// TIA Portal V16 export
// export: Created 2024-12-03T15:41:45.8171192Z, ExportSetting WithReadOnly, DisplayName Totally Integrated Automation Portal, DisplayVersion V16 Update 6, DisplayName TIA Portal Version Control Interface, DisplayVersion V16 Update 2, DisplayName TIA Portal Openness, DisplayVersion V16 Update 6, DisplayName TIA Portal Teamcenter Gateway, DisplayVersion V16, DisplayName SINAMICS Startdrive Advanced, DisplayVersion V16 Update 5, DisplayName SINAMICS Startdrive G130, G150, S120, S150, SINAMICS MV, S210, DisplayVersion V16 Update 5, DisplayName SINAMICS Startdrive G110M, G120, G120C, G120D, G120P, G115D, DisplayVersion V16 Update 5, DisplayName STEP 7 Professional, DisplayVersion V16 Update 6, DisplayName STEP 7 Safety, DisplayVersion V16, DisplayName WinCC Advanced / Unified PC, DisplayVersion V16 Update 6
TYPE "Nord_Drive_SK5xx_In_Data_UDT"
// stored: CreationDate 2024-12-03T06:55:59.9692037Z, InterfaceModifiedDate 2023-12-19T13:50:46.5922924Z, IsConsistent true, LibraryConformanceStatus The object is library-conformant., ModifiedDate 2023-12-19T13:50:46.5922924Z
   STRUCT
      MotorRunningOnSetpoint : Bool;   // 1 = Setpoint bereikt
      BusControllerActive : Bool;   // 1 = Bus controller actief
      Function4809 : Bool;   // P481 Not Used
      MotorIsRunningRight : Bool;   // 1 = Motor draait rechstom
      MotorIsRunningLeft : Bool;   // 1 = Motor draait linksom
      Function4810_MovementDone : Bool;   // P481 Not Used
      ParameterSetLsB : Bool;   // 0 = Par set 1 / 1 = Par set 2 / 2 = Par set 3 / 3 = Par set 4
      ParameterSetMSB : Bool;   // 0 = Par set 1 / 1 = Par set 2 / 2 = Par set 3 / 3 = Par set 4
      ReadyToStart : Bool;   // 1 = Ready to start
      ReadyForOperation : Bool;   // 1 = Ready for operation
      Running : Bool;   // 1 = Operation enabled
      ErrorActive : Bool;   // 1 = Drive in fout
      PowerOn : Bool;   // 0 = OFF 2 commando is uitgevoerd
      EmergencyStoPActive : Bool;   // 0 = OFF 3 commando is uitgevoerd
      CannotStartError : Bool;   // 1 = Starten niet mogelijk
      WarningActive : Bool;   // 1 = Er is een warning op de drive
      ActualSpeed : Int;   // Actual motor speed (RPM) | scale factor = 11.66
      DigitalInputs : Struct   // digital inputs
         Spare_5 : Byte;
         Input_1 : Bool;   // Digital Input 1
         Input_2 : Bool;   // Digital Input 2
         Input_3 : Bool;   // Digital Input 3
         Input_4 : Bool;   // Digital Input 4
         Input_5 : Bool;   // Digital Input 5
         Input_6 : Bool;   // Digital Input 6
         Spare_3 : Bool;
         Spare_4 : Bool;
      END_STRUCT;
      ActualCurrent : Int;   // Actual motor phase current | scale factor = 19113.33
      ErrorNumber : Int;   // Active error | 0 = no error
      ActualSetpointFrequency : Int;   // Actual setpoint frequency stator | scale factor = 327.56
   END_STRUCT;
END_TYPE
